// TIA Portal V21 export
// export: Created 2026-09-06T16:14:48.8260729Z, ExportSetting WithDefaults, DisplayName Totally Integrated Automation Portal, DisplayVersion V21 Hotfix 1, DisplayName STEP 7 Professional, DisplayVersion V21, DisplayName STEP 7 CFC, DisplayVersion V21, DisplayName STEP 7 Safety, DisplayVersion V21, DisplayName Tech WebApplication, DisplayVersion V21, DisplayName WinCC Basic/Comfort/Advanced, DisplayVersion V21, DisplayName SIMATIC Visualization Architect, DisplayVersion V21, DisplayName WinCC Unified, DisplayVersion V21, DisplayName SIMATIC Visualization Architect, DisplayVersion V21
VAR_GLOBAL   // PLC tag table "Entradas_Expansao3_SM1221"
   S20_COMP AT %I6.0 : Bool;   // Sensor de Proximidade Adicional 20 do Compactador
   S21_COMP AT %I6.1 : Bool;   // Sensor de Proximidade Adicional 21 do Compactador
   STOP6_GERAL AT %I6.2 : Bool;   // Paragem Local / Botao Cogumelo de Paragem Geral (Contacto NF)
   RESERVA_I6_5 AT %I6.5 : Bool;   // Reserva Tecnica Modulo DI 3
   RESERVA_I6_6 AT %I6.6 : Bool;   // Reserva Tecnica Modulo DI 3
   RESERVA_I6_7 AT %I6.7 : Bool;   // Reserva Tecnica Modulo DI 3
   RESERVA_I7_0 AT %I7.0 : Bool;   // Reserva Tecnica Modulo DI 3
   RESERVA_I7_1 AT %I7.1 : Bool;   // Reserva Tecnica Modulo DI 3
   RESERVA_I7_2 AT %I7.2 : Bool;   // Reserva Tecnica Modulo DI 3
   RESERVA_I7_3 AT %I7.3 : Bool;   // Reserva Tecnica Modulo DI 3
   RESERVA_I7_4 AT %I7.4 : Bool;   // Reserva Tecnica Modulo DI 3
   RESERVA_I7_5 AT %I7.5 : Bool;   // Reserva Tecnica Modulo DI 3
   RESERVA_I7_6 AT %I7.6 : Bool;   // Reserva Tecnica Modulo DI 3
   RESERVA_I7_7 AT %I7.7 : Bool;   // Reserva Tecnica Modulo DI 3
   NA_STOP_COMP AT %I6.3 : Bool;   // Botao / Paragem Local de Seguranca do Compactador
   RESERVA_I6_4 AT %I6.4 : Bool;   // Reserva Tecnica Modulo DI 3
END_VAR
